// TwinCAT 3 PLC project MemRingBuffer
// ProgramVersion: 3.1.4023.0
// libraries:
//   Tc2_Standard, * (Beckhoff Automation GmbH)
//   Tc2_System, * (Beckhoff Automation GmbH)
//   Tc2_Utilities, * (Beckhoff Automation GmbH)
//   Tc3_Module, * (Beckhoff Automation GmbH)
// project tree:
//   DUTs/ E_EventType.TcDUT, ST_Event.TcDUT
//   / PlcTask.TcTTO
//   POUs/ FB_EventBuffer.TcPOU, MAIN.TcPOU
// (motion and I/O tree: see PLC project untitled1)
// real-time tasks:
//   TASK PlcTask: cycle T#10ms, priority 20, ADS port 350
//   TASK PlcTask1: cycle T#10ms, priority 21, ADS port 351

CONFIGURATION MemRingBuffer
    RESOURCE PLC ON TwinCAT3
        TASK PlcTask(INTERVAL := T#10ms, PRIORITY := 21);
        PROGRAM MAIN WITH PlcTask : MAIN;
    END_RESOURCE
END_CONFIGURATION

// ---- DUTs/E_EventType.TcDUT
{attribute 'qualified_only'}
{attribute 'strict'}
{attribute 'to string'}
TYPE E_EventType :
(
	Alarm,
	Message
);
END_TYPE

// ---- DUTs/ST_Event.TcDUT
TYPE ST_Event :
STRUCT
	eEventType: E_EventType;
	eEventSeverity: TcEventSeverity;
	nEventIdentity: UDINT;
	sEventText: STRING(255);
	dtTimeStamp: DT;
END_STRUCT
END_TYPE

// ---- POUs/MAIN.TcPOU
PROGRAM MAIN
VAR
	Eventbuffer: FB_EventBuffer;
	
	AddEvent: BOOL;
	stEventToAdd: ST_Event;
	bEventToAddError: BOOL;
	
	
ReadAndRemoveEvent: BOOL;
stLastReadEvent: ST_Event;

bReadAndRemoveEventError:BOOL;
	nCount: UDINT;
	 
END_VAR

IF AddEvent THEN
	Eventbuffer.AddEvent(stEvent:=stEventToAdd, bError=> bEventToAddError, nCount=> nCount);
	AddEvent:= FALSE;
	
END_IF

IF ReadAndRemoveEvent THEN
		Eventbuffer.GetAndRemoveEvent(stEvent=>stLastReadEvent, bError=> bReadAndRemoveEventError, nCount=> nCount);
ReadAndRemoveEvent:=FALSE;
END_IF

IF StartNotePad THEN
	notepadStart(c
END_IF

END_PROGRAM

// ---- POUs/FB_EventBuffer.TcPOU
FUNCTION_BLOCK FB_EventBuffer

VAR
	MemRingBuffer: FB_MemRingBuffer;
	BufferArray: ARRAY[0..NUMBER_OF_BYTES_FOR_ALL_ST_EVENT] OF BYTE; //Buffer memory used BY FB_MemRingBuffer FUNCTION block
	
END_VAR

VAR CONSTANT
	SIZE_OF_ST_EVENT: UDINT:= SIZEOF(ST_Event);
    MAX_NUMBER_OF_ST_EVENTS:UDINT:=5;
	NUMBER_OF_BYTES_FOR_ALL_ST_EVENT: UDINT :=SIZE_OF_ST_EVENT * MAX_NUMBER_OF_ST_EVENTS;
	
END_VAR

METHOD AddEvent : BOOL
VAR_INPUT
	stEvent: REFERENCE TO ST_Event;
	
END_VAR

VAR_OUTPUT
	bError: BOOL;
	nCount: UDINT;
	
END_VAR
MemRingBuffer.A_AddTail(pWrite:= ADR(stEvent), 
	cbWrite:=SIZEOF(stEvent),
	pBuffer:=ADR(BufferArray),
	cbBuffer:= SIZEOF(BufferArray));
	
	bError:= NOT MemRingBuffer.bOk;
		nCount:= MemRingBuffer.nCount;
END_METHOD

METHOD GetAndRemoveEvent 
VAR_OUTPUT
	stEvent: ST_Event;
	nCount: UDINT;
	bError: BOOL;
END_VAR


	MemRingBuffer.A_RemoveHead(pRead:= ADR(stEvent), 
	cbRead:=SIZEOF(stEvent),
	pBuffer:=ADR(BufferArray),
	cbBuffer:= SIZEOF(BufferArray)); //,nCount=>nCount
	
	bError:= NOT MemRingBuffer.bOk;
			nCount:= MemRingBuffer.nCount;
END_METHOD

END_FUNCTION_BLOCK
